(* Schneider Machine Expert - Basic project Project1_Part1A, file version 1.6.0.0 *)
(* ProjectInformations: Name=New project *)

HARDWARE
  Cpu 0: TM221M16R/G
  EthernetConfiguration: NetworkName=M221, IpAllocationMode=FixedAddress, IpAddress=0.0.0.0, SubnetMask=0.0.0.0
  SerialLineConfiguration: Baud=Baud19200, Parity=ParityEven, DataBits=DataBits8, StopBits=StopBits1, PhysicalMedium=PhysicalMediumRs485, TransmissionMode=TransmissionModeModbusRtu, SlaveId=1, Addressing=SlaveAddressing
  MastTask: UsePeriodScanMode=false, PeriodScan=100
  FastTask: Period=255
  CpuBehavior: StartingMode=StartAsPreviousState, AutoSaveRamOnEeprom=true, WatchdogPeriod=250

SYMBOLS  (address, symbol, comment, settings)
  %I0.0       "Input 0"

POU New POU
  (* SectionNumber=1 *)

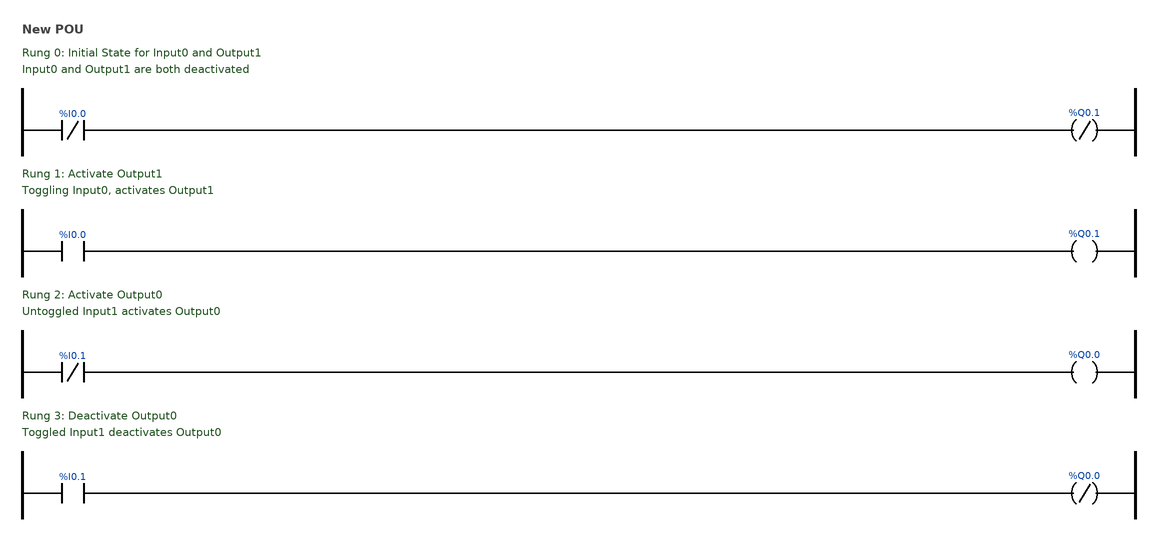

// Rung 0: Initial State for Input0 and Output1
// Input0 and Output1 are both deactivated
  LDN %I0.0
  STN %Q0.1
  // as ST:
  //   %Q0.1 := NOT (NOT %I0.0);

// Rung 1: Activate Output1
// Toggling Input0, activates Output1
  LD %I0.0
  ST %Q0.1
  // as ST:
  //   %Q0.1 := %I0.0;

// Rung 2: Activate Output0
// Untoggled Input1 activates Output0
  LDN %I0.1
  ST %Q0.0
  // as ST:
  //   %Q0.0 := NOT %I0.1;

// Rung 3: Deactivate Output0
// Toggled Input1 deactivates Output0
  LD %I0.1
  STN %Q0.0
  // as ST:
  //   %Q0.0 := NOT %I0.1;
